Yaskawa INFORM job: R2_W53-A2(90,90)(Z_REKI)AWOK.JBI

/JOB
//NAME R2_W53-A2(90,90)(Z_REKI)AWOK
///FOLDERNAME AWOK
//POS
///NPOS 51,51,0,2,0,0
///TOOL 0
///POSTYPE PULSE
///PULSE
C00000=125464,54795,11916,11,80425,-11658
C00001=121244,44056,18593,6759,72401,-26825
C00002=121230,46639,38017,7289,61852,-27463
C00003=122241,53153,48068,7083,58944,-27260
C00004=122994,55656,52047,6863,57731,-27040
C00005=122980,57562,54200,6894,57389,-27067
C00006=122635,56026,52462,7013,57691,-27185
C00007=115735,75335,76366,23767,62426,-33932
C00008=116402,75107,76087,23601,62287,-33691
C00009=115735,75335,76366,23767,62426,-33932
C00010=122958,70240,66479,6151,63242,-27072
C00011=122958,71102,68653,6199,62352,-27121
C00012=122949,71417,67723,6164,63083,-27086
C00013=122579,68264,62659,6197,64599,-27143
C00014=121633,61461,51491,6314,68030,-27307
C00015=120725,86942,86965,-6360,96130,703
C00016=120725,94594,101296,-6306,91272,948
C00017=120458,94130,102513,-6356,90267,909
C00018=120720,91828,98455,-6309,91597,931
C00019=120722,104658,115687,-6298,87608,1131
C00020=120725,93954,102220,-6300,90380,994
C00021=120725,94590,101320,-6306,91255,949
C00022=120725,86929,86977,-6360,96117,703
C00023=120724,66094,58037,-4026,59743,-41882
C00024=120724,68322,64308,-4142,57035,-41781
C00025=121179,56850,55435,-4680,51165,-41345
C00026=120602,68569,64801,-4100,56853,-41823
C00027=120553,66518,62749,-4070,57059,-41850
C00028=122230,56905,55497,-5227,51220,-40897
C00029=120724,67441,61892,-5047,61541,-36174
C00030=120724,65441,55931,-4933,64172,-36290
C00031=120746,51662,14371,-4516,82609,-36995
C00032=145452,77818,44713,-11922,79884,-28597
C00033=156803,-4554,-21296,-38868,71085,-35796
C00034=145388,-53117,-46253,-49880,51520,-42437
C00035=150930,-4046,-2869,-57376,87012,-30567
C00036=153863,24819,24400,-61587,106099,-23539
C00037=146924,20502,28447,-59274,98703,-22584
C00038=144263,18847,29999,-58387,95867,-22218
C00039=141947,-406,14710,-60739,85177,-25031
C00040=141719,1448,17330,-60050,86083,-17288
C00041=141210,-455,15065,-60828,84595,-25059
C00042=141032,770,15718,-60833,84600,-25181
C00043=140006,424,16470,-60248,85030,-17586
C00044=141965,-1146,16183,-62420,84073,-23333
C00045=144263,18847,29999,-58387,95867,-22218
C00046=147131,21787,26629,-58450,99560,-23103
C00047=150293,-4284,-1564,-60683,85300,-29337
C00048=145388,-53117,-46253,-49880,51520,-42437
C00049=145387,-55319,-59295,-46172,56236,-45294
C00050=70536,-76246,-94484,-49862,51525,-42441
BC00000=79590,232785,1075173
BC00001=74772,214348,1075175
BC00002=74772,214348,1075175
BC00003=74772,214348,1075175
BC00004=74772,214348,1075171
BC00005=74772,214348,1075171
BC00006=74772,214348,1075175
BC00007=74772,214348,1075175
BC00008=74772,214348,1075175
BC00009=74772,214348,1075175
BC00010=74772,214348,1075175
BC00011=74772,214348,1075175
BC00012=74772,214348,1075175
BC00013=74772,214348,1075175
BC00014=74772,214348,1075175
BC00015=38069,173629,1075175
BC00016=38985,172975,1075175
BC00017=39349,172746,1075174
BC00018=39352,172713,1075175
BC00019=39352,172713,1075175
BC00020=46883,172703,1075175
BC00021=46517,172965,1075175
BC00022=45600,173619,1075175
BC00023=55686,222877,1075175
BC00024=53159,219722,1075175
BC00025=52148,218460,1075175
BC00026=52148,218460,1075175
BC00027=52148,218460,1075175
BC00028=52148,218460,1075175
BC00029=47332,215529,1075175
BC00030=49711,218850,1075175
BC00031=49711,218850,1075175
BC00032=49711,218850,1075175
BC00033=17908,152957,1075175
BC00034=15,115884,1075175
BC00035=15,115884,1075175
BC00036=15,115884,1075175
BC00037=15,115884,1075175
BC00038=15,115884,1075175
BC00039=15,116385,1075175
BC00040=15,116065,1075172
BC00041=15,115443,1075175
BC00042=15,115443,1075175
BC00043=15,116065,1075172
BC00044=15,116065,1075172
BC00045=15,115884,1075175
BC00046=15,115884,1075175
BC00047=15,115884,1075175
BC00048=15,115884,1075175
BC00049=76033,260645,1075171
BC00050=76033,376048,1075171
///POSTYPE BASE
///RECTAN
///RCONF 0,0,0,0,0,0,0,0,0,0,0,0,0,0,0,0,0,0,0,0,0,0,0,0
P00006=0.222,-3.123,-1.508,0.0000,0.0000,0.0000
P00022=0.222,-3.123,-1.508,0.0000,0.0000,0.0000
//INST
///DATE 2023/11/16 10:52
///ATTR SC,RW
///GROUP1 RB1,BS1
NOP
'r2_W53-A2(90,90)(z_reki)
'Path S980
SFTOF
MOVJ C00000 BC00000 VJ=20.00
MOVJ C00001 BC00001 VJ=20.00
MOVJ C00002 BC00002 VJ=20.00
MOVL C00003 BC00003 V=100.0
MOVL C00004 BC00004 V=60.0
REFP 3 C00005 BC00005
CALL JOB:SEARCH-R1
SET P022 P006
SFTON P022
MOVL C00006 BC00006 V=60.0
MOVL C00007 BC00007 V=60.0
REFP 3 C00008 BC00008
CALL JOB:SEARCH-R1
SET P022 P006
SFTON P022
MOVL C00009 BC00009 V=60.0
MOVL C00010 BC00010 V=60.0
REFP 3 C00011 BC00011
CALL JOB:SEARCH-R1
SET P022 P006
SFTON P022
MOVL C00012 BC00012 V=60.0
MOVL C00013 BC00013 V=100.0
MOVL C00014 BC00014 V=100.0
'Path W981
SFTOF
SFTON P022
MOVL C00015 BC00015 V=100.0
MOVL C00016 BC00016 V=100.0
MOVL C00017 BC00017 V=100.0 PL=0
REFP 1 C00018 BC00018
REFP 2 C00019 BC00019
MACRO1 MJ#(0) ARGF10
ARCON
MOVL C00020 BC00020 V=10.8
ARCOF
MOVL C00021 BC00021 V=100.0
MOVL C00022 BC00022 V=100.0
SFTOF
'Path W982
SFTOF
SFTON P022
MOVJ C00023 BC00023 VJ=20.00
MOVL C00024 BC00024 V=100.0
MOVL C00025 BC00025 V=100.0 PL=0
REFP 1 C00026 BC00026
REFP 2 C00027 BC00027
MACRO1 MJ#(0) ARGF9
ARCON
MOVL C00028 BC00028 V=10.0
ARCOF
MOVL C00029 BC00029 V=100.0
MOVL C00030 BC00030 V=100.0
SFTOF
'Path VIA1071
SFTOF
MOVJ C00031 BC00031 VJ=20.00
'Path VIA1072
SFTOF
MOVJ C00032 BC00032 VJ=20.00
'Path VIA1070
SFTOF
MOVJ C00033 BC00033 VJ=20.00
MOVJ C00034 BC00034 VJ=20.00
'Path VIA1073
SFTOF
MOVJ C00035 BC00035 VJ=20.00
MOVJ C00036 BC00036 VJ=20.00
'Path VIA1069
SFTOF
'Path VIA1067
SFTOF
MOVJ C00037 BC00037 VJ=20.00
MOVJ C00038 BC00038 VJ=20.00
'Path W983
SFTOF
SFTON P022
MOVL C00039 BC00039 V=100.0
MOVL C00040 BC00040 V=100.0 PL=0
REFP 1 C00041 BC00041
REFP 2 C00042 BC00042
MACRO1 MJ#(0) ARGF9
ARCON
MOVL C00043 BC00043 V=11.7
ARCOF
MOVL C00044 BC00044 V=100.0
SFTOF
'Path VIA1063
SFTOF
MOVJ C00045 BC00045 VJ=20.00
'Path VIA1064
SFTOF
MOVJ C00046 BC00046 VJ=20.00
'Path VIA1065
SFTOF
MOVJ C00047 BC00047 VJ=20.00
'Path VIA1066
SFTOF
MOVJ C00048 BC00048 VJ=20.00
'COMMENT
MOVJ C00049 BC00049 VJ=20.00
MOVJ C00050 BC00050 VJ=20.00
END
